{attribute 'qualified_only'}
{attribute 'strict'}
TYPE E_COLD_START_STATE :
(
	NULL := 0,
	N2_PURGE,
	TEMPERATURE,	
	PRESSURISE,
	H2_PURGE
);
END_TYPE

(* stored: Version 1.1.0.1, ProductVersion 3.1.4024.12
   DUT E_COLD_START_STATE: Id {0f5a9dc1-8256-49d4-a4be-ca60beca3476} *)
